{attribute 'qualified_only'}
{attribute 'strict'}
{attribute 'to_string'}
TYPE E_MOVER_SELECTOR :
(
	SELECT_MOVER_INDEX,
  SELECT_MOVER_AXIS_ID
);
END_TYPE

(* stored: Version 1.1.0.1, ProductVersion 3.1.4026.18
   DUT E_MOVER_SELECTOR: Id {df5df385-c351-4158-9997-dc969f6ec0b8} *)
